(* IEC 61131-3 sources: JaccoSigma/tempclass/Class/ConnObjChannel, 1 file *)

(* ---- ConnObjChannel.st ---- *)
(*!
<Class
	Name               = "ConnObjChannel"
	Revision           = "0.0"
	RealtimeTask       = "false"
	CyclicTask         = "true"
	DefCyclictime      = "10 ms"
	BackgroundTask     = "false"
	Sigmatek           = "false"
	OSInterface        = "false"
	HighPriority       = "false"
	Automatic          = "false"
	UpdateMode         = "Prescan"
	SharedCommandTable = "true"
	Objectsize         = "(284,120)">
	<Channels>
		<Server Name="ClassSvr" Visualized="false" Initialize="false" WriteProtected="true" Retentive="false"/>
		<Server Name="ConnTo" Visualized="false" Initialize="false" WriteProtected="false" Retentive="false"/>
		<Server Name="State" Visualized="false" Initialize="false" WriteProtected="true" Retentive="false"/>
		<Client Name="ObjChan" Required="false" Internal="false"/>
	</Channels>
</Class>
*)
ConnObjChannel : CLASS
  //Servers:
	ClassSvr 	: SvrChCmd_DINT;
	ConnTo 	: SvrCh_DINT;
	State 	: SvrCh_DINT;
  //Clients:
	ObjChan 	: CltChCmd_MyObject;
  //Variables:
		RetCode 	: DINT;
  //Functions:

	FUNCTION VIRTUAL GLOBAL CyWork
		VAR_INPUT
			EAX 	: UDINT;
		END_VAR
		VAR_OUTPUT
			state (EAX) 	: UDINT;
		END_VAR;

	FUNCTION VIRTUAL GLOBAL ConnTo::Write
		VAR_INPUT
			input (EAX) 	: DINT;
		END_VAR
		VAR_OUTPUT
			result (EAX) 	: DINT;
		END_VAR;
  //Tables:
	FUNCTION @STD
		VAR_OUTPUT
			ret_code	: CONFSTATES;
		END_VAR;
	FUNCTION GLOBAL TAB @CT_;
END_CLASS;

#pragma usingLtd MyObject

(*
 * state
 *         0  => OK
 *        -2  => Invalid ToNr
 *        -3  => Invalid return from "ConnectCltSvr()"
 *
 *)

FUNCTION VIRTUAL GLOBAL ConnObjChannel::ConnTo::Write
	VAR_INPUT
		input (EAX) 	: DINT;
	END_VAR
	VAR_OUTPUT
		result (EAX) 	: DINT;
	END_VAR

	ConnTo := input;
  case ConnTo of
  1:
    RetCode := ConnectCltSvr( pCltName := "ConnObjChannel.ObjChan", pSvrName := "MyObject1.ClassSvr");
    if RetCode<> 1 then state  := -3; end_if;
  2:
    RetCode := ConnectCltSvr( pCltName := "ConnObjChannel.ObjChan", pSvrName := "MyObject2.ClassSvr");
    if RetCode<> 1 then state  := -3; end_if;
  3:
    RetCode := ConnectCltSvr( pCltName := "ConnObjChannel.ObjChan", pSvrName := "MyObject3.ClassSvr");
    if RetCode<> 1 then state  := -3; end_if;
  else
    State := -2;
  end_case;
 	result := ConnTo;

END_FUNCTION

FUNCTION VIRTUAL GLOBAL ConnObjChannel::CyWork
	VAR_INPUT
		EAX 	: UDINT;
	END_VAR
	VAR_OUTPUT
		state (EAX) 	: UDINT;
	END_VAR

  if IsClientConnected( #ObjChan) then
    ClassSvr  := ObjChan.AddValue( 123);
  end_if;
	state := READY;

END_FUNCTION
